(* IEC 61131-3 sources: nanopb_ST/iec61131/runtime/br/NanoPbSt, 8 files *)

(* ---- Types.typ ---- *)
(* nanoPB Runtime Library for B&R Automation Studio *)
(* nanoPB types ported to B&R IEC 61131-3 ST *)
(* Basic data type for storing encoded data and other byte streams *)

TYPE
	pb_byte_t : USINT; (* Data type for storing sizes of struct fields and array counts *)
	pb_size_t : UINT;
	pb_ssize_t : INT; (* Field type information - encodes field type, allocation and repetition *)
	pb_type_t : USINT; (* Wire types for protocol buffer encoding *)
	pb_wire_type_t :
		( (* 64-bit unsigned integer structure for B&R compatibility *)
		PB_WT_VARINT := 0,
		PB_WT_64BIT := 1,
		PB_WT_STRING := 2,
		PB_WT_32BIT := 5
		);
	pb_uint64_struct : 	STRUCT
		low : UDINT; (* Lower 32 bits *)
		high : UDINT; (* Upper 32 bits *)
	END_STRUCT;
END_TYPE

(* Input stream structure for decoding *)

TYPE
	pb_istream_struct : 	STRUCT  (* Callback function would go here - not applicable in B&R *) (* We'll use buffer-only mode *) (* Free field for implementation use *)
		state : REFERENCE TO UDINT; (* Buffer pointer and remaining bytes *)
		bytes_left : pb_size_t; (* Error message for debugging *)
		errmsg : STRING[80];
	END_STRUCT;
END_TYPE

(* Output stream structure for encoding *)

TYPE
	pb_ostream_struct : 	STRUCT  (* Free field for implementation use *)
		state : REFERENCE TO UDINT; (* Buffer pointer and size limits *)
		max_size : pb_size_t;
		bytes_written : pb_size_t; (* Error message for debugging *)
		errmsg : STRING[80];
	END_STRUCT;
END_TYPE

(* Message descriptor - describes the fields in a message *)

TYPE
	pb_msgdesc_struct : 	STRUCT  (* Field information array *)
		field_info : REFERENCE TO UDINT; (* Array of encoded field descriptors *) (* Submessage descriptors *)
		submsg_info : REFERENCE TO UDINT; (* Array of pointers to pb_msgdesc_struct *) (* Default values *)
		default_value : REFERENCE TO pb_byte_t; (* Field counts and metadata *)
		callback : UDINT;
		field_count : pb_size_t;
		required_field_count : pb_size_t;
		largest_tag : pb_size_t;
	END_STRUCT;
END_TYPE

(* Field iterator for processing message fields *)

TYPE
	pb_field_iter_struct : 	STRUCT  (* Message descriptor *)
		descriptor : REFERENCE TO pb_msgdesc_struct; (* Current message being processed *)
		message : REFERENCE TO UDINT; (* void* equivalent *) (* Iterator state *)
		index : pb_size_t;
		field_info_index : pb_size_t;
		required_field_index : pb_size_t;
		submessage_index : pb_size_t; (* Current field information *)
		tag : pb_size_t;
		data_size : pb_size_t;
		array_size : pb_size_t;
		type : pb_type_t; (* Pointers to current field data *)
		pField : REFERENCE TO UDINT;
		pData : REFERENCE TO UDINT;
		pSize : REFERENCE TO UDINT; (* For submessages *)
		submsg_desc : REFERENCE TO pb_msgdesc_struct;
	END_STRUCT;
END_TYPE

(* Byte array structure - variable length data *)

TYPE
	pb_bytes_array_struct : 	STRUCT
		size : pb_size_t;
		bytes : ARRAY[0..0]OF pb_byte_t; (* Will be larger in practice *)
	END_STRUCT;
END_TYPE

(* ---- NanoPbSt.fun ---- *)
(* nanoPB Runtime Library for B&R Automation Studio *)
(* nanoPB library functions ported to B&R IEC 61131-3 ST *)
(* ===== STREAM FUNCTIONS ===== *)

FUNCTION pb_st_istream_from_buffer : UDINT (*Create input stream from buffer - returns address*) (*$GROUP=nanoPB,$CAT=Stream,$GROUPICON=User.png,$CATICON=User.png*)
	VAR_INPUT
		stream : pb_istream_struct; (* Stream to initialize *)
		buf : REFERENCE TO pb_byte_t; (* Buffer containing data *)
		bufsize : pb_size_t; (* Size of buffer *)
	END_VAR
END_FUNCTION

FUNCTION pb_st_ostream_from_buffer : UDINT (*Create output stream from buffer - returns address*) (*$GROUP=nanoPB,$CAT=Stream,$GROUPICON=User.png,$CATICON=User.png*)
	VAR_INPUT
		stream : pb_ostream_struct; (* Stream to initialize *)
		buf : REFERENCE TO pb_byte_t; (* Buffer to write to *)
		bufsize : pb_size_t; (* Size of buffer *)
	END_VAR
END_FUNCTION

FUNCTION pb_st_read : BOOL (*Read data from input stream*) (*$GROUP=nanoPB,$CAT=Stream,$GROUPICON=User.png,$CATICON=User.png*)
	VAR_INPUT
		stream : pb_istream_struct; (* Input stream *)
		buf : UDINT; (* Buffer to read into *)
		count : pb_size_t; (* Number of bytes to read *)
	END_VAR
	VAR
		i : pb_size_t;
		src_ptr : REFERENCE TO pb_byte_t;
		dest_ptr : REFERENCE TO pb_byte_t;
	END_VAR
END_FUNCTION

FUNCTION pb_st_write : BOOL (*Write data to output stream*) (*$GROUP=nanoPB,$CAT=Stream,$GROUPICON=User.png,$CATICON=User.png*)
	VAR_INPUT
		stream : pb_ostream_struct; (* Output stream *)
		buf : UDINT; (* Buffer to write from *)
		count : pb_size_t; (* Number of bytes to write *)
	END_VAR
	VAR
		i : pb_size_t;
		src_ptr : REFERENCE TO pb_byte_t;
		dest_ptr : REFERENCE TO pb_byte_t;
	END_VAR
END_FUNCTION
(* ===== VARINT FUNCTIONS ===== *)

FUNCTION pb_st_encode_varint : BOOL (*Encode unsigned varint*) (*$GROUP=nanoPB,$CAT=Varint,$GROUPICON=User.png,$CATICON=User.png*)
	VAR_INPUT
		stream : pb_ostream_struct; (* Output stream *)
		value : UDINT; (* Value to encode *)
	END_VAR
	VAR
		buffer : ARRAY[0..9] OF pb_byte_t; (* Max 10 bytes for 64-bit varint *)
		i : USINT;
		bytes_written : USINT;
	END_VAR
END_FUNCTION

FUNCTION pb_st_decode_varint : BOOL (*Decode unsigned varint*) (*$GROUP=nanoPB,$CAT=Varint,$GROUPICON=User.png,$CATICON=User.png*)
	VAR_INPUT
		stream : pb_istream_struct; (* Input stream *)
		dest : REFERENCE TO UDINT; (* Destination for decoded value *)
	END_VAR
	VAR
		byte_val : pb_byte_t;
		bitpos : USINT;
		result : UDINT;
	END_VAR
END_FUNCTION

FUNCTION pb_st_encode_svarint : BOOL (*Encode signed varint (zigzag)*) (*$GROUP=nanoPB,$CAT=Varint,$GROUPICON=User.png,$CATICON=User.png*)
	VAR_INPUT
		stream : pb_ostream_struct; (* Output stream *)
		value : DINT; (* Signed value to encode *)
	END_VAR
	VAR
		encoded : UDINT;
	END_VAR
END_FUNCTION

FUNCTION pb_st_decode_svarint : BOOL (*Decode signed varint (zigzag)*) (*$GROUP=nanoPB,$CAT=Varint,$GROUPICON=User.png,$CATICON=User.png*)
	VAR_INPUT
		stream : pb_istream_struct; (* Input stream *)
		dest : REFERENCE TO DINT; (* Destination for decoded value *)
	END_VAR
	VAR
		encoded : UDINT;
	END_VAR
END_FUNCTION
(* ===== FIELD ENCODING/DECODING ===== *)

FUNCTION pb_st_encode_tag_for_field : BOOL (*Encode field tag and wire type*) (*$GROUP=nanoPB,$CAT=Field,$GROUPICON=User.png,$CATICON=User.png*)
	VAR_INPUT
		stream : pb_ostream_struct; (* Output stream *)
		field : pb_field_iter_struct; (* Field iterator *)
	END_VAR
	VAR
		wire_type : USINT;
		tag_and_type : UDINT;
		length : UDINT;
	END_VAR
END_FUNCTION

FUNCTION pb_st_encode_string : BOOL (*Encode string field*) (*$GROUP=nanoPB,$CAT=Field,$GROUPICON=User.png,$CATICON=User.png*)
	VAR_INPUT
		stream : pb_ostream_struct; (* Output stream *)
		s : REFERENCE TO STRING[80]; (* String to encode *)
	END_VAR
	VAR
		str_len : pb_size_t;
	END_VAR
END_FUNCTION

FUNCTION pb_st_decode_string : BOOL (*Decode string field*) (*$GROUP=nanoPB,$CAT=Field,$GROUPICON=User.png,$CATICON=User.png*)
	VAR_INPUT
		stream : pb_istream_struct; (* Input stream *)
		dest : REFERENCE TO STRING[80]; (* Destination string *)
		size : pb_size_t; (* Maximum string size *)
	END_VAR
	VAR
		str_len : UDINT;
		temp_str : STRING[255];
	END_VAR
END_FUNCTION

FUNCTION pb_st_encode_fixed32 : BOOL (*Encode 32-bit fixed field*) (*$GROUP=nanoPB,$CAT=Field,$GROUPICON=User.png,$CATICON=User.png*)
	VAR_INPUT
		stream : pb_ostream_struct; (* Output stream *)
		value : UDINT; (* Value to encode *)
	END_VAR
	VAR
		bytes : ARRAY[0..3] OF pb_byte_t;
	END_VAR
END_FUNCTION

FUNCTION pb_st_decode_fixed32 : BOOL (*Decode 32-bit fixed field*) (*$GROUP=nanoPB,$CAT=Field,$GROUPICON=User.png,$CATICON=User.png*)
	VAR_INPUT
		stream : pb_istream_struct; (* Input stream *)
		dest : REFERENCE TO UDINT; (* Destination for value *)
	END_VAR
	VAR
		bytes : ARRAY[0..3] OF pb_byte_t;
	END_VAR
END_FUNCTION

FUNCTION pb_st_encode_fixed64 : BOOL (*Encode 64-bit fixed field*) (*$GROUP=nanoPB,$CAT=Field,$GROUPICON=User.png,$CATICON=User.png*)
	VAR_INPUT
		stream : pb_ostream_struct; (* Output stream *)
		value : pb_uint64_struct; (* Value to encode *)
	END_VAR
	VAR
		bytes : ARRAY[0..7] OF pb_byte_t;
		i : USINT;
	END_VAR
END_FUNCTION

FUNCTION pb_st_decode_fixed64 : BOOL (*Decode 64-bit fixed field*) (*$GROUP=nanoPB,$CAT=Field,$GROUPICON=User.png,$CATICON=User.png*)
	VAR_INPUT
		stream : pb_istream_struct; (* Input stream *)
		dest : REFERENCE TO pb_uint64_struct; (* Destination for value *)
	END_VAR
	VAR
		bytes : ARRAY[0..7] OF pb_byte_t;
		i : USINT;
	END_VAR
END_FUNCTION
(* ===== FIELD ITERATOR FUNCTIONS ===== *)

FUNCTION pb_st_field_iter_begin : BOOL (*Initialize field iterator*) (*$GROUP=nanoPB,$CAT=Iterator,$GROUPICON=User.png,$CATICON=User.png*)
	VAR_INPUT
		iter : pb_field_iter_struct; (* Iterator to initialize *)
		descriptor : pb_msgdesc_struct; (* Message descriptor *)
		message : UDINT; (* Message structure *)
	END_VAR
END_FUNCTION

FUNCTION pb_st_field_iter_next : BOOL (*Move to next field*) (*$GROUP=nanoPB,$CAT=Iterator,$GROUPICON=User.png,$CATICON=User.png*)
	VAR_INPUT
		iter : pb_field_iter_struct; (* Field iterator *)
	END_VAR
	VAR
		desc_ref : REFERENCE TO pb_msgdesc_struct;
		field_info_ptr : REFERENCE TO ARRAY[0..0] OF UDINT;
		prev_descriptor : UDINT;
		descriptor_len : UDINT;
		prev_type : USINT;
	END_VAR
END_FUNCTION

FUNCTION pb_st_field_iter_find : BOOL (*Find field by tag*) (*$GROUP=nanoPB,$CAT=Iterator,$GROUPICON=User.png,$CATICON=User.png*)
	VAR_INPUT
		iter : pb_field_iter_struct; (* Field iterator *)
		tag : pb_size_t; (* Tag to find *)
	END_VAR
	VAR
		dpb_msgdesc_struct : REFERENCE TO pb_msgdesc_struct;
	END_VAR
END_FUNCTION
(* ===== MAIN ENCODE/DECODE FUNCTIONS ===== *)

FUNCTION pb_st_encode : BOOL (*Encode message to stream*) (*$GROUP=nanoPB,$CAT=Main,$GROUPICON=User.png,$CATICON=User.png*)
	VAR_INPUT
		stream : pb_ostream_struct; (* Output stream *)
		fields : pb_msgdesc_struct; (* Message descriptor *)
		src_struct : UDINT; (* Source message structure *)
	END_VAR
	VAR
		iter : pb_field_iter_struct;
		iter_ref : REFERENCE TO pb_field_iter_struct;
	END_VAR
END_FUNCTION

FUNCTION pb_st_decode : BOOL (*Decode message from stream*) (*$GROUP=nanoPB,$CAT=Main,$GROUPICON=User.png,$CATICON=User.png*)
	VAR_INPUT
		stream : pb_istream_struct; (* Input stream *)
		fields : pb_msgdesc_struct; (* Message descriptor *)
		dest_struct : UDINT; (* Destination message structure *)
	END_VAR
	VAR
		tag : UDINT;
		wire_type : pb_wire_type_t;
		tag_value : pb_size_t;
		iter : pb_field_iter_struct;
		iter_ref : REFERENCE TO pb_field_iter_struct;
		field_found : BOOL;
	END_VAR
END_FUNCTION
(* ===== UTILITY FUNCTIONS ===== *)

FUNCTION pb_st_skip_field : BOOL (*Skip unknown field based on wire type*) (*$GROUP=nanoPB,$CAT=Utility,$GROUPICON=User.png,$CATICON=User.png*)
	VAR_INPUT
		stream : pb_istream_struct; (* Input stream *)
		wire_type : pb_wire_type_t; (* Wire type of field to skip *)
	END_VAR
	VAR
		length : UDINT;
		dummy_value : UDINT;
		dummy_value64 : pb_uint64_struct;
	END_VAR
END_FUNCTION

FUNCTION pb_st_make_string_substream : BOOL (*Create substream for string/bytes*) (*$GROUP=nanoPB,$CAT=Utility,$GROUPICON=User.png,$CATICON=User.png*)
	VAR_INPUT
		stream : pb_istream_struct; (* Input stream *)
		substream : pb_istream_struct; (* Substream to create *)
	END_VAR
	VAR
		length : UDINT;
	END_VAR
END_FUNCTION

FUNCTION pb_st_close_string_substream : BOOL (*Close string/bytes substream*) (*$GROUP=nanoPB,$CAT=Utility,$GROUPICON=User.png,$CATICON=User.png*)
	VAR_INPUT
		stream : pb_istream_struct; (* Original stream *)
		substream : pb_istream_struct; (* Substream to close *)
	END_VAR
END_FUNCTION
(* ===== INTERNAL HELPER FUNCTIONS ===== *)

FUNCTION pb_st_load_descriptor_values : BOOL (*Load field descriptor values*) (*$GROUP=nanoPB,$CAT=Internal,$GROUPICON=User.png,$CATICON=User.png*)
	VAR_INPUT
		iter : pb_field_iter_struct; (* Field iterator *)
	END_VAR
	VAR
		desc_ref : REFERENCE TO pb_msgdesc_struct;
		word0 : UDINT;
		word1 : UDINT;
		word2 : UDINT;
		word3 : UDINT;
		word4 : UDINT;
		data_offset : UDINT;
		size_offset : DINT;
		size_offset_raw : UDINT;
		descriptor_format : UDINT;
		field_info_ptr : REFERENCE TO ARRAY[0..0] OF UDINT;
		ptr_ptr : REFERENCE TO UDINT;
	END_VAR
END_FUNCTION

FUNCTION pb_st_encode_field : BOOL (*Encode single field*) (*$GROUP=nanoPB,$CAT=Internal,$GROUPICON=User.png,$CATICON=User.png*)
	VAR_INPUT
		stream : pb_ostream_struct; (* Output stream *)
		field : pb_field_iter_struct; (* Field iterator *)
	END_VAR
	VAR
		field_type : USINT;
		has_value : BOOL;
		bool_ptr : REFERENCE TO BOOL;
		int_ptr : REFERENCE TO DINT;
		uint_ptr : REFERENCE TO UDINT;
		real_ptr : REFERENCE TO REAL;
		val_64 : REFERENCE TO pb_uint64_struct;
		string_ptr : REFERENCE TO STRING[80];
	END_VAR
END_FUNCTION

FUNCTION pb_st_decode_field : BOOL (*Decode single field*) (*$GROUP=nanoPB,$CAT=Internal,$GROUPICON=User.png,$CATICON=User.png*)
	VAR_INPUT
		stream : pb_istream_struct; (* Input stream *)
		field : pb_field_iter_struct; (* Field iterator *)
		wire_type : pb_wire_type_t; (* Wire type from tag *)
	END_VAR
	VAR
		field_type : USINT;
		expected_wire_type : pb_wire_type_t;
		temp_uint : UDINT;
		bool_ptr : REFERENCE TO BOOL;
	END_VAR
END_FUNCTION

FUNCTION pb_st_init_default_values : BOOL (*Initialize message with defaults*) (*$GROUP=nanoPB,$CAT=Internal,$GROUPICON=User.png,$CATICON=User.png*)
	VAR_INPUT
		fields : pb_msgdesc_struct; (* Message descriptor *)
		dest_struct : REFERENCE TO UDINT; (* Message structure *)
	END_VAR
END_FUNCTION

(* ---- pb_codec.st ---- *)
(* nanoPB Runtime Library for B&R Automation Studio *)
(* nanoPB main encode/decode functions *)
(* Ported from nanoPB C library to B&R IEC 61131-3 ST *)

FUNCTION pb_st_encode

	iter_ref ACCESS ADR(iter);

	(* Initialize field iterator *)
	IF NOT pb_st_field_iter_begin(iter_ref, fields, src_struct) THEN
		pb_st_encode := TRUE; (* Empty message is valid *)
		RETURN;
	END_IF;

	(* Encode all fields *)
	REPEAT
		IF NOT pb_st_encode_field(stream, iter_ref) THEN
			pb_st_encode := FALSE;
			RETURN;
		END_IF;
	UNTIL NOT pb_st_field_iter_next(iter_ref) END_REPEAT;

	pb_st_encode := TRUE;

END_FUNCTION

FUNCTION pb_st_decode

	iter_ref ACCESS ADR(iter);

	(* Initialize message with default values *)
	pb_st_init_default_values(fields, dest_struct);

	(* Decode fields until end of stream *)
	WHILE stream.bytes_left > 0 DO
		(* Read field tag and wire type *)
		IF NOT pb_st_decode_varint(stream, ADR(tag)) THEN
			pb_st_decode := FALSE;
			RETURN;
		END_IF;

		(* Extract wire type (3 lowest bits) and tag (remaining bits) *)
		wire_type := UDINT_TO_USINT(tag AND 16#07);
		tag_value := UDINT_TO_UINT(SHR(tag, 3));

		(* Find field descriptor *)
		field_found := pb_st_field_iter_begin(iter_ref, fields, dest_struct);
		IF field_found THEN
			field_found := pb_st_field_iter_find(iter_ref, tag_value);
		END_IF;

		IF field_found THEN
			(* Decode known field *)
			IF NOT pb_st_decode_field(stream, iter_ref, wire_type) THEN
				pb_st_decode := FALSE;
				RETURN;
			END_IF;
		ELSE
			(* Skip unknown field *)
			IF NOT pb_st_skip_field(stream, wire_type) THEN
				pb_st_decode := FALSE;
				RETURN;
			END_IF;
		END_IF;
	END_WHILE;

	pb_st_decode := TRUE;

END_FUNCTION

FUNCTION pb_st_encode_field

	field_type := field.type AND PB_LTYPE_MASK;

	(* Check if field has a value (for optional fields) *)
	has_value := TRUE;
	IF (field.type AND PB_HTYPE_MASK) = PB_HTYPE_OPTIONAL THEN
		IF field.pSize <> 0 THEN
			bool_ptr ACCESS field.pSize;
			has_value := bool_ptr;
		END_IF;
	END_IF;

	IF NOT has_value THEN
		pb_st_encode_field := TRUE; (* Skip optional field without value *)
		RETURN;
	END_IF;

	(* Encode field tag and wire type *)
	IF NOT pb_st_encode_tag_for_field(stream, field) THEN
		pb_st_encode_field := FALSE;
		RETURN;
	END_IF;

	(* Encode field value based on type *)
	CASE field_type OF
		PB_LTYPE_BOOL:
			bool_ptr ACCESS field.pData;
			IF bool_ptr THEN
				pb_st_encode_field := pb_st_encode_varint(stream, 1);
			ELSE
				pb_st_encode_field := pb_st_encode_varint(stream, 0);
			END_IF;

		PB_LTYPE_VARINT, PB_LTYPE_UVARINT:
			uint_ptr ACCESS field.pData;
			pb_st_encode_field := pb_st_encode_varint(stream, uint_ptr);

		PB_LTYPE_SVARINT:
			int_ptr ACCESS field.pData;
			pb_st_encode_field := pb_st_encode_svarint(stream, int_ptr);

		PB_LTYPE_FIXED32:
			uint_ptr ACCESS field.pData;
			pb_st_encode_field := pb_st_encode_fixed32(stream, uint_ptr);

		PB_LTYPE_FIXED64:
			val_64 ACCESS field.pData;
			pb_st_encode_field := pb_st_encode_fixed64(stream, val_64);

		PB_LTYPE_STRING:
			string_ptr ACCESS field.pData;
			pb_st_encode_field := pb_st_encode_string(stream, ADR(string_ptr));

	ELSE
		stream.errmsg := PB_ERR_INVALID_FIELD;
		pb_st_encode_field := FALSE;
	END_CASE;

END_FUNCTION

FUNCTION pb_st_decode_field

	field_type := field.type AND PB_LTYPE_MASK;

	(* Determine expected wire type *)
	CASE field_type OF
		PB_LTYPE_BOOL, PB_LTYPE_VARINT, PB_LTYPE_UVARINT, PB_LTYPE_SVARINT:
			expected_wire_type := PB_WT_VARINT;
		PB_LTYPE_FIXED32:
			expected_wire_type := PB_WT_32BIT;
		PB_LTYPE_FIXED64:
			expected_wire_type := PB_WT_64BIT;
		PB_LTYPE_STRING, PB_LTYPE_BYTES:
			expected_wire_type := PB_WT_STRING;
	ELSE
		stream.errmsg := PB_ERR_INVALID_FIELD;
		pb_st_decode_field := FALSE;
		RETURN;
	END_CASE;

	(* Check wire type matches *)
	IF wire_type <> expected_wire_type THEN
		stream.errmsg := PB_ERR_INVALID_WIRE_TYPE;
		pb_st_decode_field := FALSE;
		RETURN;
	END_IF;

	(* Decode field value based on type *)
	CASE field_type OF
		PB_LTYPE_BOOL:
			IF pb_st_decode_varint(stream, ADR(temp_uint)) THEN
				bool_ptr ACCESS field.pData;
				bool_ptr := (temp_uint <> 0);
				pb_st_decode_field := TRUE;
			ELSE
				pb_st_decode_field := FALSE;
			END_IF;

		PB_LTYPE_VARINT, PB_LTYPE_UVARINT:
			pb_st_decode_field := pb_st_decode_varint(stream, field.pData);

		PB_LTYPE_SVARINT:
			pb_st_decode_field := pb_st_decode_svarint(stream, field.pData);

		PB_LTYPE_FIXED32:
			pb_st_decode_field := pb_st_decode_fixed32(stream, field.pData);

		PB_LTYPE_FIXED64:
			pb_st_decode_field := pb_st_decode_fixed64(stream, field.pData);

		PB_LTYPE_STRING:
			pb_st_decode_field := pb_st_decode_string(stream, field.pData, 255);

	ELSE
		stream.errmsg := PB_ERR_INVALID_FIELD;
		pb_st_decode_field := FALSE;
	END_CASE;

	(* Set has_field flag for optional fields *)
	IF pb_st_decode_field AND ((field.type AND PB_HTYPE_MASK) = PB_HTYPE_OPTIONAL) THEN
		IF field.pSize <> 0 THEN
			bool_ptr ACCESS field.pSize;
			bool_ptr := TRUE;
		END_IF;
	END_IF;

END_FUNCTION

FUNCTION pb_st_init_default_values

	(* For now, just zero out the entire structure *)
	(* In a full implementation, this would set proper default values *)
//	brsmemset(dest_struct, 0, 1024); (* Assume max 1KB message size *)
	pb_st_init_default_values := TRUE;

END_FUNCTION

(* ---- pb_fields.st ---- *)
(* nanoPB Runtime Library for B&R Automation Studio *)
(* nanoPB field encoding/decoding functions *)
(* Ported from nanoPB C library to B&R IEC 61131-3 ST *)

FUNCTION pb_st_encode_tag_for_field

	(* Determine wire type based on field type *)
	CASE (field.type AND PB_LTYPE_MASK) OF
		PB_LTYPE_BOOL, PB_LTYPE_VARINT, PB_LTYPE_UVARINT, PB_LTYPE_SVARINT:
			wire_type := DINT_TO_USINT(PB_WT_VARINT);
		PB_LTYPE_FIXED32:
			wire_type := DINT_TO_USINT(PB_WT_32BIT);
		PB_LTYPE_FIXED64:
			wire_type := DINT_TO_USINT(PB_WT_64BIT);
		PB_LTYPE_STRING, PB_LTYPE_BYTES, PB_LTYPE_SUBMESSAGE, PB_LTYPE_FIXED_LENGTH_BYTES:
			wire_type := DINT_TO_USINT(PB_WT_STRING);
	ELSE
		stream.errmsg := PB_ERR_INVALID_FIELD;
		pb_st_encode_tag_for_field := FALSE;
		RETURN;
	END_CASE;

	(* Combine tag and wire type: (tag << 3) | wire_type *)
	tag_and_type := SHL(UINT_TO_UDINT(field.tag), 3) OR USINT_TO_UDINT(wire_type);

	pb_st_encode_tag_for_field := pb_st_encode_varint(stream, tag_and_type);

END_FUNCTION

FUNCTION pb_st_encode_fixed32

	(* Encode as little-endian 32-bit *)
	bytes[0] := UDINT_TO_USINT(value AND 16#FF);
	bytes[1] := UDINT_TO_USINT(SHR(value, 8) AND 16#FF);
	bytes[2] := UDINT_TO_USINT(SHR(value, 16) AND 16#FF);
	bytes[3] := UDINT_TO_USINT(SHR(value, 24) AND 16#FF);

	pb_st_encode_fixed32 := pb_st_write(stream, ADR(bytes[0]), 4);

END_FUNCTION

FUNCTION pb_st_decode_fixed32

	IF NOT pb_st_read(stream, ADR(bytes[0]), 4) THEN
		pb_st_decode_fixed32 := FALSE;
		RETURN;
	END_IF;

	(* Decode from little-endian 32-bit *)
	dest := USINT_TO_UDINT(bytes[0]) OR
	         SHL(USINT_TO_UDINT(bytes[1]), 8) OR
	         SHL(USINT_TO_UDINT(bytes[2]), 16) OR
	         SHL(USINT_TO_UDINT(bytes[3]), 24);

	pb_st_decode_fixed32 := TRUE;

END_FUNCTION

FUNCTION pb_st_encode_fixed64

	(* Encode as little-endian 64-bit from structure *)
	(* Encode lower 32 bits *)
	FOR i := 0 TO 3 DO
		bytes[i] := UDINT_TO_USINT(SHR(value.low, i * 8) AND 16#FF);
	END_FOR;

	(* Encode upper 32 bits *)
	FOR i := 4 TO 7 DO
		bytes[i] := UDINT_TO_USINT(SHR(value.high, (i - 4) * 8) AND 16#FF);
	END_FOR;

	pb_st_encode_fixed64 := pb_st_write(stream, ADR(bytes[0]), 8);

END_FUNCTION

FUNCTION pb_st_decode_fixed64

	IF NOT pb_st_read(stream, ADR(bytes[0]), 8) THEN
		pb_st_decode_fixed64 := FALSE;
		RETURN;
	END_IF;

	(* Decode from little-endian 64-bit into structure *)
	dest.low := 0;
	dest.high := 0;

	(* Decode lower 32 bits *)
	FOR i := 0 TO 3 DO
		dest.low := dest.low OR SHL(USINT_TO_UDINT(bytes[i]), i * 8);
	END_FOR;

	(* Decode upper 32 bits *)
	FOR i := 4 TO 7 DO
		dest.high := dest.high OR SHL(USINT_TO_UDINT(bytes[i]), (i - 4) * 8);
	END_FOR;

	pb_st_decode_fixed64 := TRUE;

END_FUNCTION

FUNCTION pb_st_encode_string

	str_len := UDINT_TO_UINT(brsstrlen(ADR(s)));

	(* First encode the string length as varint *)
	IF NOT pb_st_encode_varint(stream, UINT_TO_UDINT(str_len)) THEN
		pb_st_encode_string := FALSE;
		RETURN;
	END_IF;

	(* Then encode the string bytes *)
	pb_st_encode_string := pb_st_write(stream, ADR(s), str_len);

END_FUNCTION

FUNCTION pb_st_decode_string

	(* First decode the string length *)
	IF NOT pb_st_decode_varint(stream, ADR(str_len)) THEN
		pb_st_decode_string := FALSE;
		RETURN;
	END_IF;

	(* Check if string fits in destination *)
	IF str_len >= size THEN
		stream.errmsg := PB_ERR_BUFFER_OVERFLOW;
		pb_st_decode_string := FALSE;
		RETURN;
	END_IF;

	(* Read string bytes *)
	IF str_len > 0 THEN
		IF NOT pb_st_read(stream, ADR(temp_str), UDINT_TO_UINT(str_len)) THEN
			pb_st_decode_string := FALSE;
			RETURN;
		END_IF;

		(* Null terminate and copy to destination *)
		brsmemcpy(ADR(dest), ADR(temp_str), UDINT_TO_UINT(str_len));
	END_IF;

	pb_st_decode_string := TRUE;

END_FUNCTION

FUNCTION pb_st_skip_field

	CASE wire_type OF
		PB_WT_VARINT:
			(* Skip varint by reading and discarding *)
			pb_st_skip_field := pb_st_decode_varint(stream, ADR(dummy_value));

		PB_WT_32BIT:
			(* Skip 4 bytes *)
			pb_st_skip_field := pb_st_decode_fixed32(stream, ADR(dummy_value));

		PB_WT_64BIT:
			(* Skip 8 bytes *)
			pb_st_skip_field := pb_st_decode_fixed64(stream, ADR(dummy_value64));

		PB_WT_STRING:
			(* Read length and skip that many bytes *)
			IF pb_st_decode_varint(stream, ADR(length)) THEN
				IF stream.bytes_left >= UDINT_TO_UINT(length) THEN
					stream.state := stream.state + UDINT_TO_UINT(length);
					stream.bytes_left := stream.bytes_left - UDINT_TO_UINT(length);
					pb_st_skip_field := TRUE;
				ELSE
					stream.errmsg := PB_ERR_EOF;
					pb_st_skip_field := FALSE;
				END_IF;
			ELSE
				pb_st_skip_field := FALSE;
			END_IF;

	ELSE
		stream.errmsg := PB_ERR_INVALID_WIRE_TYPE;
		pb_st_skip_field := FALSE;
	END_CASE;

END_FUNCTION

(* ---- pb_iterator.st ---- *)
(* nanoPB Runtime Library for B&R Automation Studio *)
(* nanoPB field iterator functions *)
(* Ported from nanoPB C library to B&R IEC 61131-3 ST *)

FUNCTION pb_st_field_iter_begin

	(* Initialize field iterator *)
	iter.descriptor := ADR(descriptor);
	iter.message := message;
	iter.index := 0;
	iter.field_info_index := 0;
	iter.required_field_index := 0;
	iter.submessage_index := 0;

	(* Load first field if it exists *)
	IF descriptor.field_count > 0 THEN
		pb_st_field_iter_begin := pb_st_load_descriptor_values(iter);
	ELSE
		pb_st_field_iter_begin := FALSE;
	END_IF;

END_FUNCTION

FUNCTION pb_st_field_iter_next

	(* Move to next field *)
	iter.index := iter.index + 1;

	desc_ref ACCESS iter.descriptor;
	IF iter.index >= desc_ref.field_count THEN
		pb_st_field_iter_next := FALSE;
		RETURN;
	END_IF;

	(* Increment field_info_index based on previous field descriptor format *)
	(* Get the previous field descriptor to determine its length *)
	field_info_ptr ACCESS desc_ref.field_info;
	prev_descriptor := field_info_ptr[iter.field_info_index];

	(* Calculate descriptor length: 2^(lowest 2 bits) words *)
	descriptor_len := SHL(1, (prev_descriptor AND 16#03));

	(* Advance field_info_index by descriptor length *)
	iter.field_info_index := iter.field_info_index + UDINT_TO_UINT(descriptor_len);

	(* Update other indexes if needed *)
	prev_type := UDINT_TO_USINT(SHR(prev_descriptor, 8) AND 16#FF);
	IF (prev_type AND PB_HTYPE_MASK) = PB_HTYPE_REQUIRED THEN
		iter.required_field_index := iter.required_field_index + 1;
	END_IF;

	(* Load values for the new field *)
	pb_st_field_iter_next := pb_st_load_descriptor_values(iter);

END_FUNCTION

FUNCTION pb_st_field_iter_find

	(* Reset to beginning *)
	dpb_msgdesc_struct ACCESS iter.descriptor;
	IF NOT pb_st_field_iter_begin(iter, dpb_msgdesc_struct, iter.message) THEN
		pb_st_field_iter_find := FALSE;
		RETURN;
	END_IF;

	(* Search for matching tag *)
	REPEAT
		IF iter.tag = tag THEN
			pb_st_field_iter_find := TRUE;
			RETURN;
		END_IF;
	UNTIL NOT pb_st_field_iter_next(iter) END_REPEAT;

	pb_st_field_iter_find := FALSE;

END_FUNCTION

FUNCTION pb_st_load_descriptor_values

	desc_ref ACCESS iter.descriptor;
	IF iter.index >= desc_ref.field_count THEN
		pb_st_load_descriptor_values := FALSE;
		RETURN;
	END_IF;

	(* Get the field info array and access the current field descriptor *)
	field_info_ptr ACCESS desc_ref.field_info;
	word0 := field_info_ptr[iter.field_info_index];

	(* Extract field type - always in bits 8-15 *)
	iter.type := UDINT_TO_USINT(SHR(word0, 8) AND 16#FF);

	(* Handle different descriptor formats based on lowest 2 bits *)
	descriptor_format := word0 AND 16#03;

	CASE descriptor_format OF
		0: (* 1-word format *)
			(* Tag is in bits 2-7 *)
			iter.tag := UDINT_TO_UINT(SHR(word0, 2) AND 16#3F);
			(* Size offset is in bits 24-27 (signed 4-bit) *)
			size_offset_raw := SHR(word0, 24) AND 16#0F;
			IF size_offset_raw >= 8 THEN
				size_offset := UDINT_TO_DINT(size_offset_raw) - 16;
			ELSE
				size_offset := UDINT_TO_DINT(size_offset_raw);
			END_IF;
			(* Data offset is in bits 16-23 *)
			data_offset := SHR(word0, 16) AND 16#FF;
			(* Data size is in bits 28-31 *)
			iter.data_size := UDINT_TO_UINT(SHR(word0, 28) AND 16#0F);
			(* Array size is 1 for single fields *)
			iter.array_size := 1;

		1: (* 2-word format *)
			word1 := field_info_ptr[iter.field_info_index + 1];
			(* Array size is in bits 16-27 of word0 *)
			iter.array_size := UDINT_TO_UINT(SHR(word0, 16) AND 16#0FFF);
			(* Tag combines bits 2-7 of word0 and bits 28-31 of word1 *)
			iter.tag := UDINT_TO_UINT((SHR(word0, 2) AND 16#3F) OR (SHR(word1, 28) * 64));
			(* Size offset is in bits 28-31 of word0 (signed 4-bit) *)
			size_offset_raw := SHR(word0, 28) AND 16#0F;
			IF size_offset_raw >= 8 THEN
				size_offset := UDINT_TO_DINT(size_offset_raw) - 16;
			ELSE
				size_offset := UDINT_TO_DINT(size_offset_raw);
			END_IF;
			(* Data offset is in bits 0-15 of word1 *)
			data_offset := word1 AND 16#FFFF;
			(* Data size is in bits 16-27 of word1 *)
			iter.data_size := UDINT_TO_UINT(SHR(word1, 16) AND 16#0FFF);

		2: (* 4-word format *)
			word1 := field_info_ptr[iter.field_info_index + 1];
			word2 := field_info_ptr[iter.field_info_index + 2];
			word3 := field_info_ptr[iter.field_info_index + 3];
			(* Array size is in bits 16-31 of word0 *)
			iter.array_size := UDINT_TO_UINT(SHR(word0, 16));
			(* Tag combines bits 2-7 of word0 and bits 8-31 of word1 *)
			iter.tag := UDINT_TO_UINT((SHR(word0, 2) AND 16#3F) OR (SHR(word1, 8) * 64));
			(* Size offset is in bits 0-7 of word1 (signed 8-bit) *)
			size_offset_raw := word1 AND 16#FF;
			IF size_offset_raw >= 128 THEN
				size_offset := UDINT_TO_DINT(size_offset_raw) - 256;
			ELSE
				size_offset := UDINT_TO_DINT(size_offset_raw);
			END_IF;
			(* Data offset is word2 *)
			data_offset := word2;
			(* Data size is word3 *)
			iter.data_size := UDINT_TO_UINT(word3);

		3: (* 8-word format *)
			word1 := field_info_ptr[iter.field_info_index + 1];
			word2 := field_info_ptr[iter.field_info_index + 2];
			word3 := field_info_ptr[iter.field_info_index + 3];
			word4 := field_info_ptr[iter.field_info_index + 4];
			(* Array size is word4 *)
			iter.array_size := UDINT_TO_UINT(word4);
			(* Tag combines bits 2-7 of word0 and bits 8-31 of word1 *)
			iter.tag := UDINT_TO_UINT((SHR(word0, 2) AND 16#3F) OR (SHR(word1, 8) * 64));
			(* Size offset is in bits 0-7 of word1 (signed 8-bit) *)
			size_offset_raw := word1 AND 16#FF;
			IF size_offset_raw >= 128 THEN
				size_offset := UDINT_TO_DINT(size_offset_raw) - 256;
			ELSE
				size_offset := UDINT_TO_DINT(size_offset_raw);
			END_IF;
			(* Data offset is word2 *)
			data_offset := word2;
			(* Data size is word3 *)
			iter.data_size := UDINT_TO_UINT(word3);

	END_CASE;

	(* Calculate field pointers *)
	IF iter.message = 0 THEN
		(* Avoid arithmetic on null pointers *)
		iter.pField := 0;
		iter.pSize := 0;
		iter.pData := 0;
	ELSE
		iter.pField := iter.message + data_offset;

		(* Calculate pSize based on size_offset from nanoPB descriptor *)
		IF size_offset <> 0 THEN
			(* Standard nanoPB format with explicit size_offset *)
			iter.pSize := UDINT_TO_DINT(iter.pField) - size_offset;
		ELSIF (iter.type AND PB_HTYPE_MASK) = PB_HTYPE_REPEATED AND
			  ((iter.type AND PB_ATYPE_MASK) = PB_ATYPE_STATIC OR (iter.type AND PB_ATYPE_MASK) = PB_ATYPE_POINTER) THEN
			(* For repeated fields, pSize points to array_size *)
			iter.pSize := ADR(iter.array_size);
		ELSE
			(* Required/singular fields don't need size field *)
			iter.pSize := 0;
		END_IF;

		(* Calculate pData based on allocation type *)
		IF (iter.type AND PB_ATYPE_MASK) = PB_ATYPE_POINTER AND iter.pField <> 0 THEN
			(* For pointer fields, pData is the pointed-to location *)
			ptr_ptr ACCESS iter.pField;
			iter.pData := ptr_ptr;
		ELSE
			(* For static allocation, pData same as pField *)
			iter.pData := iter.pField;
		END_IF;
	END_IF;

	pb_st_load_descriptor_values := TRUE;

END_FUNCTION

(* ---- pb_stream.st ---- *)
(* nanoPB Runtime Library for B&R Automation Studio *)
(* nanoPB stream functions *)
(* Ported from nanoPB C library to B&R IEC 61131-3 ST *)

FUNCTION pb_st_istream_from_buffer

	(* Initialize input stream from buffer *)
	stream.state := ADR(buf); (* Store buffer pointer in state *)
	stream.bytes_left := bufsize;
	stream.errmsg := '';

	pb_st_istream_from_buffer := ADR(stream);

END_FUNCTION

FUNCTION pb_st_ostream_from_buffer

	(* Initialize output stream from buffer *)
	stream.state := ADR(buf); (* Store buffer pointer in state *)
	stream.max_size := bufsize;
	stream.bytes_written := 0;
	stream.errmsg := '';

	pb_st_ostream_from_buffer := ADR(stream);

END_FUNCTION

FUNCTION pb_st_read

	(* Check if we have enough bytes *)
	IF stream.bytes_left < count THEN
		stream.errmsg := PB_ERR_EOF;
		pb_st_read := FALSE;
		RETURN;
	END_IF;

	(* Copy bytes from stream buffer to destination *)
	src_ptr ACCESS stream.state;
	dest_ptr ACCESS buf;

	(* Use platform memory copy function for efficient memory copying *)
	brsmemcpy(ADR(dest_ptr), ADR(src_ptr), count);

	(* Update stream position *)
	stream.state := stream.state + count;
	stream.bytes_left := stream.bytes_left - count;

	pb_st_read := TRUE;

END_FUNCTION

FUNCTION pb_st_write

	(* Check if we have enough space *)
	IF stream.bytes_written + count > stream.max_size THEN
		stream.errmsg := PB_ERR_BUFFER_OVERFLOW;
		pb_st_write := FALSE;
		RETURN;
	END_IF;

	(* Copy bytes from source to stream buffer *)
	(* Use platform memory copy function for efficient memory copying *)
	brsmemcpy(stream.state, buf, count);
	stream.state := stream.state + count;
	(* Update stream position *)
	stream.bytes_written := stream.bytes_written + count;

	pb_st_write := TRUE;

END_FUNCTION

FUNCTION pb_st_make_string_substream

	(* First decode the string length *)
	IF NOT pb_st_decode_varint(stream, ADR(length)) THEN
		pb_st_make_string_substream := FALSE;
		RETURN;
	END_IF;

	(* Check if we have enough data *)
	IF stream.bytes_left < UDINT_TO_UINT(length) THEN
		stream.errmsg := PB_ERR_EOF;
		pb_st_make_string_substream := FALSE;
		RETURN;
	END_IF;

	(* Initialize substream from current position *)
	substream.state := stream.state;
	substream.bytes_left := UDINT_TO_UINT(length);
	substream.errmsg := '';

	(* Advance main stream *)
	stream.state := stream.state + UDINT_TO_UINT(length);
	stream.bytes_left := stream.bytes_left - UDINT_TO_UINT(length);

	pb_st_make_string_substream := TRUE;

END_FUNCTION

FUNCTION pb_st_close_string_substream

	(* Skip any remaining bytes in substream *)
	IF substream.bytes_left > 0 THEN
		substream.state := substream.state + substream.bytes_left;
		substream.bytes_left := 0;
	END_IF;

	pb_st_close_string_substream := TRUE;

END_FUNCTION

(* ---- pb_varint.st ---- *)
(* nanoPB Runtime Library for B&R Automation Studio *)
(* nanoPB varint encoding/decoding functions *)
(* Ported from nanoPB C library to B&R IEC 61131-3 ST *)

FUNCTION pb_st_encode_varint

	(* Encode varint using 7-bit encoding *)
	i := 0;

	REPEAT
		buffer[i] := UDINT_TO_USINT(value AND 16#7F); (* Take lower 7 bits *)
		value := SHR(value, 7); (* Shift right by 7 bits *)

		IF value <> 0 THEN
			buffer[i] := buffer[i] OR 16#80; (* Set continuation bit *)
		END_IF;

		i := i + 1;
	UNTIL value = 0 OR i >= 10 END_REPEAT;

	bytes_written := i;

	(* Write the encoded bytes to stream *)
	pb_st_encode_varint := pb_st_write(stream, ADR(buffer[0]), bytes_written);

END_FUNCTION

FUNCTION pb_st_decode_varint

	result := 0;
	bitpos := 0;

	(* Decode varint using 7-bit encoding *)
	REPEAT
		IF NOT pb_st_read(stream, ADR(byte_val), 1) THEN
			pb_st_decode_varint := FALSE;
			RETURN;
		END_IF;

		(* Add the 7 bits to result *)
		result := result OR SHL(USINT_TO_UDINT(byte_val AND 16#7F), bitpos);
		bitpos := bitpos + 7;

		(* Check if we have more bytes (continuation bit set) *)
		IF (byte_val AND 16#80) = 0 THEN
			EXIT; (* No more bytes *)
		END_IF;

		(* Prevent overflow - max 5 bytes for 32-bit value *)
		IF bitpos >= 32 THEN
			stream.errmsg := 'Varint overflow';
			pb_st_decode_varint := FALSE;
			RETURN;
		END_IF;

	UNTIL FALSE END_REPEAT;

	dest := result;
	pb_st_decode_varint := TRUE;

END_FUNCTION

FUNCTION pb_st_encode_svarint

	(* ZigZag encode: (n << 1) ^ (n >> 31) *)
	IF value >= 0 THEN
		encoded := SHL(DINT_TO_UDINT(value), 1);
	ELSE
		encoded := SHL(DINT_TO_UDINT(value), 1) XOR 16#FFFFFFFF;
	END_IF;

	pb_st_encode_svarint := pb_st_encode_varint(stream, encoded);

END_FUNCTION

FUNCTION pb_st_decode_svarint

	IF NOT pb_st_decode_varint(stream, ADR(encoded)) THEN
		pb_st_decode_svarint := FALSE;
		RETURN;
	END_IF;

	(* ZigZag decode: (n >> 1) ^ (-(n & 1)) *)
	IF (encoded AND 1) = 0 THEN
		dest := UDINT_TO_DINT(SHR(encoded, 1));
	ELSE
		dest := UDINT_TO_DINT(SHR(encoded, 1)) XOR UDINT_TO_DINT(16#FFFFFFFF);
	END_IF;

	pb_st_decode_svarint := TRUE;

END_FUNCTION

(* ---- Constants.var ---- *)
VAR CONSTANT
	(* nanoPB constants ported to B&R *)

	(* Field type constants - least significant 4 bits *)
	PB_LTYPE_BOOL : USINT := 16#00;
	PB_LTYPE_VARINT : USINT := 16#01;
	PB_LTYPE_UVARINT : USINT := 16#02;
	PB_LTYPE_SVARINT : USINT := 16#03;
	PB_LTYPE_FIXED32 : USINT := 16#04;
	PB_LTYPE_FIXED64 : USINT := 16#05;
	PB_LTYPE_BYTES : USINT := 16#06;
	PB_LTYPE_STRING : USINT := 16#07;
	PB_LTYPE_SUBMESSAGE : USINT := 16#08;
	PB_LTYPE_SUBMSG_W_CB : USINT := 16#09;
	PB_LTYPE_EXTENSION : USINT := 16#0A;
	PB_LTYPE_FIXED_LENGTH_BYTES : USINT := 16#0B;

	(* Field repetition rules *)
	PB_HTYPE_REQUIRED : USINT := 16#00;
	PB_HTYPE_OPTIONAL : USINT := 16#10;
	PB_HTYPE_SINGULAR : USINT := 16#10;
	PB_HTYPE_REPEATED : USINT := 16#20;
	PB_HTYPE_FIXARRAY : USINT := 16#20;
	PB_HTYPE_ONEOF : USINT := 16#30;

	(* Field allocation types *)
	PB_ATYPE_STATIC : USINT := 16#00;
	PB_ATYPE_POINTER : USINT := 16#80;
	PB_ATYPE_CALLBACK : USINT := 16#40;

	(* Bit masks *)
	PB_LTYPE_MASK : USINT := 16#0F;
	PB_HTYPE_MASK : USINT := 16#30;
	PB_ATYPE_MASK : USINT := 16#C0;

	(* Maximum values *)
	PB_SIZE_MAX : UINT := 65535;
	PB_MAX_REQUIRED_FIELDS : USINT := 64;

	(* Wire type constants *)
	PB_WIRE_TYPE_MASK : USINT := 16#07;

	(* nanoPB version *)
	NANOPB_VERSION : STRING[20] := 'nanopb-1.0.0-dev-B&R';

	(* Error constants *)
	PB_ERR_NONE : STRING[30] := '';
	PB_ERR_IO : STRING[30] := 'IO error';
	PB_ERR_INVALID_FIELD : STRING[30] := 'Invalid field';
	PB_ERR_INVALID_TAG : STRING[30] := 'Invalid tag';
	PB_ERR_INVALID_WIRE_TYPE : STRING[30] := 'Invalid wire type';
	PB_ERR_EOF : STRING[30] := 'End of stream';
	PB_ERR_BUFFER_OVERFLOW : STRING[30] := 'Buffer overflow';

	(* ===== SENSOR READING MESSAGE CONSTANTS ===== *)

	(* Field tags *)
	SensorReading_sensor_id_tag : USINT := 1;
	SensorReading_temperature_tag : USINT := 2;
	SensorReading_alarm_active_tag : USINT := 3;

	(* Maximum encoded message size *)
	SensorReading_size : USINT := 18;

END_VAR
